// TIA Portal V17 export
// export: Created 2024-09-15T12:29:47.9689423Z, ExportSetting WithDefaults, DisplayName Totally Integrated Automation Portal, DisplayVersion V17, DisplayName TIA Portal Openness, DisplayVersion V17, DisplayName TIA Portal Version Control Interface, DisplayVersion V17, DisplayName STEP 7 Professional, DisplayVersion V17, DisplayName STEP 7 Safety, DisplayVersion V17, DisplayName WinCC Professional, DisplayVersion V17
DATA_BLOCK "PRG_SLD_Ablauf_DB"   // DB20
AUTHOR : A.Schaefer
VERSION : 0.1
// stored: AutoNumber true, DBAccessibleFromOPCUA true, DBAccessibleFromWebserver true, InstanceOfName PRG_SLD_Ablauf, InstanceOfType FB
"PRG_SLD_Ablauf"
   // VAR
   //    lx_Init { ExternalAccessible := 'False'; ExternalVisible := 'False'; ExternalWritable := 'False'} : Bool;
   //    Location : Bool;
   //    lx_Start_TON_Wait { ExternalAccessible := 'False'; ExternalVisible := 'False'; ExternalWritable := 'False'} : Bool;
   //    lx_Time_Error { ExternalAccessible := 'False'; ExternalVisible := 'False'; ExternalWritable := 'False'} : Bool;
   //    lt_TON_Wait { ExternalAccessible := 'False'; ExternalVisible := 'False'; ExternalWritable := 'False'} : Time;
   //    lx_Start_TON_State { ExternalAccessible := 'False'; ExternalVisible := 'False'; ExternalWritable := 'False'} : Bool;
   //    ldt_MQTT { ExternalAccessible := 'False'; ExternalVisible := 'False'; ExternalWritable := 'False'} : Date_And_Time;
   //    li_Return_LDT { ExternalAccessible := 'False'; ExternalVisible := 'False'; ExternalWritable := 'False'} : Int;
   //    li_Lights { ExternalAccessible := 'False'; ExternalVisible := 'False'; ExternalWritable := 'False'} : Int;
   //    li_Lights_old { ExternalAccessible := 'False'; ExternalVisible := 'False'; ExternalWritable := 'False'} : Int;
   //    lw_ColorValueMin { ExternalAccessible := 'False'; ExternalVisible := 'False'; ExternalWritable := 'False'} : Word;
   //    li_CounterActual { ExternalAccessible := 'False'; ExternalVisible := 'False'; ExternalWritable := 'False'} : Int;
   //    lx_White { ExternalAccessible := 'False'; ExternalVisible := 'False'; ExternalWritable := 'False'} : Bool;
   //    lx_Blue { ExternalAccessible := 'False'; ExternalVisible := 'False'; ExternalWritable := 'False'} : Bool;
   //    lx_Red { ExternalAccessible := 'False'; ExternalVisible := 'False'; ExternalWritable := 'False'} : Bool;
   //    li_StepCase { ExternalAccessible := 'False'; ExternalVisible := 'False'; ExternalWritable := 'False'} : Int;
   //    ls_Color { ExternalAccessible := 'False'; ExternalVisible := 'False'; ExternalWritable := 'False'} : String;
   //    lfb_TOF_ConveyerBelt_Out { ExternalAccessible := 'False'; ExternalVisible := 'False'; ExternalWritable := 'False'} : TOF_TIME;
   //    lfb_TON_Wait { ExternalAccessible := 'False'; ExternalVisible := 'False'; ExternalWritable := 'False'} : TON_TIME;
   //    lfb_TON_Error { ExternalAccessible := 'False'; ExternalVisible := 'False'; ExternalWritable := 'False'} : TON_TIME;
   //    lfb_TON_State { ExternalAccessible := 'False'; ExternalVisible := 'False'; ExternalWritable := 'False'} : TON_TIME;
   //    lfb_F_Trig_Counter { ExternalAccessible := 'False'; ExternalVisible := 'False'; ExternalWritable := 'False'} : F_TRIG;
   //    lfb_R_Trig_Counter { ExternalAccessible := 'False'; ExternalVisible := 'False'; ExternalWritable := 'False'} : R_TRIG;
   // END_VAR
BEGIN
END_DATA_BLOCK
